(* CoDeSys 2.3.9.28 project: Aula14_ex.pro *)
(* Libraries: Standard.lib 27.1.09 11:27:38, Util.lib 27.1.09 11:27:38, IecSfc.lib 24.11.08 08:07:15, SysLibTime.lib 27.1.09 11:27:38, SysTaskInfo.lib 24.11.08 08:07:15, SYSLIBCALLBACK.LIB 27.1.09 11:27:38 *)

(* PLC configuration (modules and I/O channels)
CPX-CEC [Root] node -1, in %IB0 out %QB0 {StringParam = 2773,0,0,0,0; ByteParam = 0; ByteParam = 31; ByteParam = 0; ByteParam = 0; ByteParam = 0; ByteParam = 0; ByteParam = 0; ByteParam = 0; ByteParam = 2; ByteParam = 0; ByteParam = 0; ByteParam = 0; ByteParam = 32; ByteParam = 0; ByteParam = 0; ByteParam = 5; ByteParam = 0; ByteParam = 0; ByteParam = 0; ByteParam = 0; ByteParam = 0; ByteParam = 0; ByteParam = 0; ByteParam = 0; ByteParam = 14; ByteParam = 240; ByteParam = 192; ByteParam = 168; ByteParam = 2; ByteParam = 10; ByteParam = 255; ByteParam = 255; ByteParam = 0; ByteParam = 0; ByteParam = 192; ByteParam = 168; ByteParam = 1; ByteParam = 1; ByteParam = 192; ByteParam = 168; ByteParam = 2; ByteParam = 10; ByteParam = 255; ByteParam = 255; ByteParam = 0; ByteParam = 0; ByteParam = 192; ByteParam = 168; ByteParam = 1; ByteParam = 1}
  Hexswitch AT %IB0 [HexSwitch] rotary switch 0 = STOP, 1-15 = RUN
  IOModules [CPX_MASTER] node 0, in %IB4 out %QB0
*)

(* Global variable list: Global_Variables *)
VAR_GLOBAL

	START: BOOL;
	STOP : BOOL;
	S1: BOOL;
	S2: BOOL;
	S3: BOOL;
	FS: BOOL;
	SP: BOOL;

	LP: BOOL;
	AL: BOOL;
	EV1: BOOL;
	EV2: BOOL;
	EV3: BOOL;
	EV4: BOOL;

	MEM1 : BOOL;
	MEM2 : BOOL;
	MEM3: BOOL;
	MEM4: BOOL;

	MEMTAL: BOOL;
	MEMTEV3: BOOL;
	MEMTSTART: BOOL;
	MEMTTERMINOU: BOOL;
	MEMLAMP:BOOL;

	CONT1 : CTU;
	TV2 : TON;
	TV3 : TON;
	TV4 : TON;
	TAL : TON;
	TLAMP : TON;

END_VAR

(* POU PLC_PRG, ST *)
PROGRAM PLC_PRG
VAR
END_VAR
TV2(IN := MEM1, PT:= T#1s);
TV3(IN := MEM2, PT:= T#1s);
TV4(IN := MEM3, PT:= T#2s);
TAL(IN := MEM4, PT:= T#5s);
CONT1(CU := FS AND MEMTAL, RESET := NOT STOP OR TLAMP.Q, PV := 2);
TLAMP(IN := CONT1.Q, PT:= T#2s);

IF (START AND NOT MEMTSTART AND NOT SP) OR MEMTTERMINOU THEN
	IF NOT LP THEN
		EV1 := TRUE;
		MEMTSTART := TRUE;
		MEMTTERMINOU := FALSE;
	END_IF
END_IF

IF S1 AND EV1 THEN
	EV1 := FALSE;
	MEM1 := TRUE;
END_IF

IF TV2.Q THEN
	EV2 := TRUE;
	MEM1 := FALSE;
END_IF

IF S2 AND EV2 THEN
	EV2 := FALSE;
	MEM2 := TRUE;
END_IF

IF TV3.Q THEN
	EV3 := TRUE;
	MEM2 := FALSE;
	MEMTEV3 := TRUE;
END_IF

IF S3 AND MEMTEV3 THEN
	EV4 := TRUE;
	MEM3 := TRUE;
	MEMTAL := TRUE;
	MEMTEV3 := FALSE;
END_IF

IF FS AND MEMTAL THEN
	EV3 := FALSE;
	EV4 := FALSE;
	MEM3 := FALSE;
	MEMTAL := FALSE;
	MEMTTERMINOU := TRUE;
END_IF


IF TV4.Q AND MEM3 THEN
	MEMTTERMINOU := FALSE;
	EV3 := FALSE;
	EV4 := FALSE;
	MEM4 := TRUE;
	MEMTAL := FALSE;
	IF TAL.Q THEN
		AL := FALSE;
	ELSE
		AL := TRUE;
	END_IF
END_IF


IF CONT1.Q THEN
	IF TLAMP.Q THEN
		LP := FALSE;
	ELSE
		LP := TRUE;
	END_IF
END_IF

IF NOT STOP OR (SP AND MEMTTERMINOU) THEN
	MEMTSTART := FALSE;
	EV1 := FALSE;
	EV2 := FALSE;
	EV3 := FALSE;
	EV4 := FALSE;
	LP := FALSE;
	AL := FALSE;
	MEM1 := FALSE;
	MEM2 := FALSE;
	MEM3 := FALSE;
	MEM4 := FALSE;
	MEMTAL := FALSE;
	MEMTEV3 := FALSE;
	MEMTTERMINOU := FALSE;
END_IF
END_PROGRAM

(* Visualisation screen
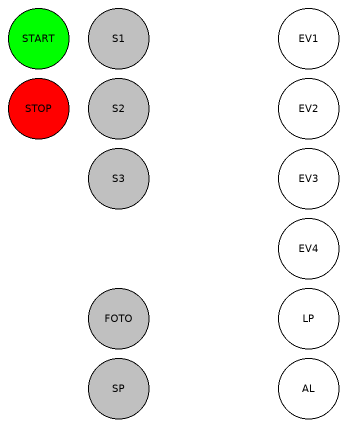
ellipse at (130,50)-(191,111): text "S1"; alarm colour if S1; taps S1
ellipse at (130,120)-(191,181): text "S2"; alarm colour if S2; taps S2
ellipse at (130,190)-(191,251): text "S3"; alarm colour if S3; taps S3
ellipse at (50,50)-(111,111): text "START"; alarm colour if START; taps START
ellipse at (50,120)-(111,181): text "STOP"; alarm colour if STOP; taps STOP
ellipse at (320,50)-(381,111): text "EV1"; alarm colour if EV1
ellipse at (320,330)-(381,391): text "LP"; alarm colour if LP
ellipse at (320,120)-(381,181): text "EV2"; alarm colour if EV2
ellipse at (320,190)-(381,251): text "EV3"; alarm colour if EV3
ellipse at (320,260)-(381,321): text "EV4"; alarm colour if EV4
ellipse at (130,330)-(191,391): text "FOTO"; alarm colour if FS; taps FS
ellipse at (130,400)-(191,461): text "SP"; alarm colour if SP; toggles SP
ellipse at (320,400)-(381,461): text "AL"; alarm colour if AL
*)
